TYPE U_CAM_DATA :
UNION
  stCtrl              : ARRAY[1..MAX_AXIS] OF ST_CAM_DATA;

  byCtrl    AT %I*    : ARRAY[1..MAX_AXIS] OF
                        ARRAY[1..SIZEOF(ST_CAM_DATA)] OF BYTE;
END_UNION
END_TYPE

(* stored: Version 1.1.0.1, ProductVersion 3.1.4026.13
   DUT U_CAM_DATA: Id {bb3adaa7-885d-4e2f-a88f-b2d8fb8017c9} *)
